PROGRAM MAIN
VAR
	Pressure_sensor : INT := 1;
	Pressure_Goal : INT := 1;	
	Pump_speed : INT := 0;
	Water_presence_sensor : BOOL;
	Water_presence_light : BOOL;
	
	Pump_on : BOOL;
	System_on : BOOL;
	System_off : BOOL;
	System_switch : BOOL;
END_VAR

IF system_switch THEN
	system_on := TRUE;
	system_off := FALSE;
ELSE
	system_on := FALSE;
	system_off := TRUE;
END_IF

IF Pressure_Goal < Pressure_sensor THEN
	IF Water_presence_sensor AND system_on THEN
		pump_on := TRUE;
	ELSE
		pump_on := FALSE;	
	END_IF
END_IF

IF water_presence_sensor THEN
	water_presence_light := TRUE;
ELSE
	water_presence_light := FALSE;
END_IF

IF Pump_on THEN
	IF Pump_speed < 100 THEN
		Pump_speed := Pump_speed + 1;
	END_IF
END_IF

IF NOT Pump_on THEN
	IF pump_speed > 1 THEN
		Pump_speed := Pump_speed - 1;
	END_IF
END_IF

END_PROGRAM

(* stored: Version 1.1.0.1, ProductVersion 3.1.4024.12
   POU MAIN: Id {07d00137-d46d-4449-9634-144601a3da1a}, SpecialFunc None *)
